(* Logix 5000 project; controller STAT 1756-L72 rev 20.12; software revision 20.04; part 12 of 34 *)
(* tags used below, declared in another part *)
   B10 : DINT[20];
   B14 : DINT[30];
   B16 : DINT[30];
   B17 : DINT[30];
   B3 : DINT[256];
   B9 : DINT[40];
   DateTime : DINT[7];   // DINT array tag for retrieve wallclock time through GSV created during conversion
   F8 : REAL[256];
   I10_000_Bit07 : ALIAS FOR I10[0].7;   // Hand Automaat CL8
   I10_000_Bit08 : ALIAS FOR I10[0].8;   // Drukknop start CL8 P 20
   I10_000_Bit09 : ALIAS FOR I10[0].9;   // Drukknop stop CL8 P 20
   I19_000_Bit02 : ALIAS FOR I19[0].2;   // vanne pmp puit 3 ouverte
   I19_000_Bit03 : ALIAS FOR I19[0].3;   // vanne pmp puit 3 fermee
   I19_000_Bit04 : ALIAS FOR I19[0].4;   // vanne pmp puit 2 ouverte
   I19_000_Bit05 : ALIAS FOR I19[0].5;   // vanne pmp puit 2 fermee
   I1_005_Bit15 : ALIAS FOR I1[5].15;
   I1_008_Bit01 : ALIAS FOR I1[8].1;   // Hand Automaat stormbekken
   I2_000_Bit04 : ALIAS FOR I2[0].4;   // Deelnoodstop cl6 eurowater
   I2_000_Bit05 : ALIAS FOR I2[0].5;   // Deelnoodstop cl7 IBT A
   I2_000_Bit07 : ALIAS FOR I2[0].7;   // Deelnoodstop cl7 IBT C
   I4_000_Bit00 : ALIAS FOR I4[0].0;   // Motor P3 voedingspomp in lijn
   I4_000_Bit03 : ALIAS FOR I4[0].3;   // Thermische storing voedingspomp fabriek 2
   I4_000_Bit04 : ALIAS FOR I4[0].4;   // Motor p4 in lijn in
   I4_000_Bit05 : ALIAS FOR I4[0].5;   // ready drive p4
   I4_000_Bit06 : ALIAS FOR I4[0].6;   // defaut drive P4
   I4_000_Bit11 : ALIAS FOR I4[0].11;   // pomp p23 in kelderkuip in dienst
   I5_001_Bit15 : ALIAS FOR I5[1].15;   // EV7_OPEN
   I6_000_Bit03 : ALIAS FOR I6[0].3;   // TH pmp PUT 2
   I6_000_Bit04 : ALIAS FOR I6[0].4;   // TH PMP PUT over
   I6_000_Bit05 : ALIAS FOR I6[0].5;   // th PMP PUT 1
   I6_000_Bit06 : ALIAS FOR I6[0].6;   // non existant th pmp 1 vijver
   I6_001_Bit04 : ALIAS FOR I6[1].4;   // niveau silo disolvent
   I7_000_Bit07 : ALIAS FOR I7[0].7;   // hoog alarm ketel tampon
   I7_000_Bit10 : ALIAS FOR I7[0].10;   // zeer hoog alarm ketel clarifee
   I7_000_Bit11 : ALIAS FOR I7[0].11;   // hoog zeer hoog alarm ketel clarifee
   I7_000_Bit12 : ALIAS FOR I7[0].12;   // laag alarm ketel clarifee
   I7_000_Bit13 : ALIAS FOR I7[0].13;   // zeer laag alarm ketel clarifee
   I7_001_Bit00 : ALIAS FOR I7[1].0;   // lus 4 niveau ketel clarifiee kontakt 3
   I9_000_Bit09 : ALIAS FOR I9[0].9;   // Hand_Auto CL7
   I9_000_Bit12 : ALIAS FOR I9[0].12;   // Drukknop start CL7 P4
   I9_000_Bit13 : ALIAS FOR I9[0].13;   // Drukknop stop CL7 P4
   I9_001_Bit00 : ALIAS FOR I9[1].0;   // Drukknop start CL7 P6
   I9_001_Bit01 : ALIAS FOR I9[1].1;   // Drukknop stop CL7 P6
   MW : BOOL;
   N11 : DINT[150];
   N12 : DINT[230];
   N13 : DINT[230];
   N7 : DINT[255];
   O12_000_Bit00 : ALIAS FOR O12[0].0;   // spoelpomp filters dubbele media P6_SPOEL
   O12_000_Bit12 : ALIAS FOR O12[0].12;   // Motor P19a zuiveringspomp controleweger P19_ZUIVERP
   O12_000_Bit13 : ALIAS FOR O12[0].13;   // Motor P20 zuiveringspomp controleweger P20_ZUIVERP
   O12_001_Bit03 : ALIAS FOR O12[1].3;   // Motor P7 voedingspomp omgekeerde osmose 1 P7_OSMOSE_1
   O12_001_Bit04 : ALIAS FOR O12[1].4;   // Motor P8 voedingspomp omgekeerde osmose 2 P8_OSMOSE_2
   O12_001_Bit05 : ALIAS FOR O12[1].5;   // Motor P9 voedingspomp omgekeerde osmose 3 P9_OSMOSE_3
   O15_001_Bit06 : ALIAS FOR O15[1].6;   // EV2 EV2
   O15_001_Bit11 : ALIAS FOR O15[1].11;   // EV7 EV7
   O16_000_Bit01 : ALIAS FOR O16[0].1;   // vanne pmp puit 3
   O16_000_Bit02 : ALIAS FOR O16[0].2;   // vanne pmp puit 2
   O18_001_Bit00 : ALIAS FOR O18[1].0;   // pompe 1 puisard ligne 4
   O18_001_Bit01 : ALIAS FOR O18[1].1;   // pompe 2 puisard ligne 4
   O18_001_Bit02 : ALIAS FOR O18[1].2;   // pmp put 2
   O18_001_Bit03 : ALIAS FOR O18[1].3;   // PMP PUT over
   O18_001_Bit04 : ALIAS FOR O18[1].4;   // PMP PUT 1
   O18_001_Bit05 : ALIAS FOR O18[1].5;   // pmp vijver IWM
   O18_001_Bit07 : ALIAS FOR O18[1].7;   // pomp pompen uit kelder p23
   O18_001_Bit08 : ALIAS FOR O18[1].8;   // pomp pompen uit kelder p24
   O1_006_Bit15 : ALIAS FOR O1[6].15;
   O27_000 : ALIAS FOR O27[0];
   O27_001 : ALIAS FOR O27[1];
   P4 : BOOL;
   Q2 : REAL;
   SCP_SPEED_PMP_FAB : SCP;
   SPEED_P3 : DINT;
   t1 : TIMER;
   T27 : TIMER[100];
   T4 : TIMER[200];
(* ibt, continued *)

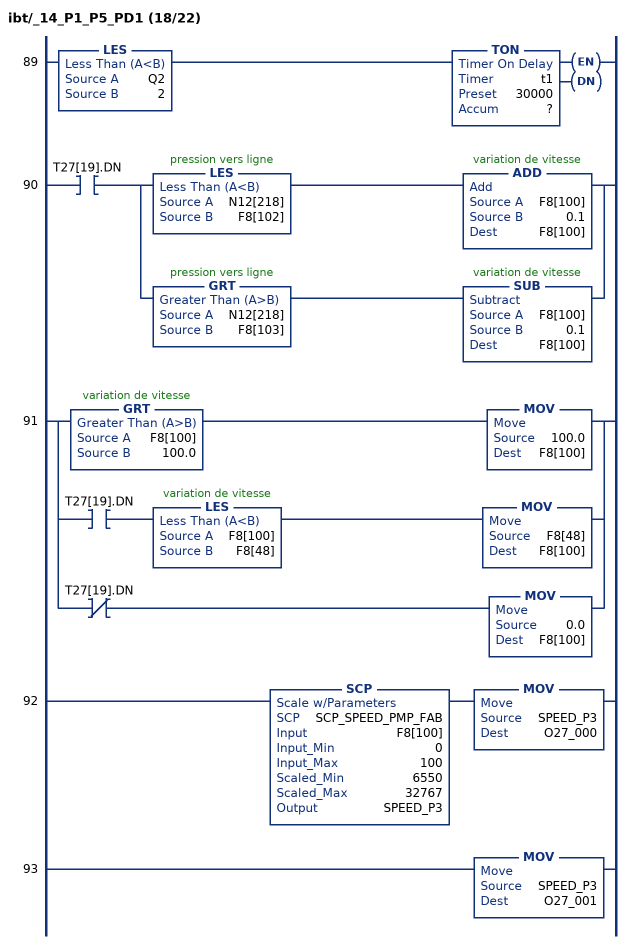
   [picture p178: ibt/_14_P1_P5_PD1 rungs 89-93]
   89: LES(Q2,2)TON(t1,?,?);
   90: XIC(T27[19].DN)[LES(N12[218],F8[102]) ADD(F8[100],0.1,F8[100]) ,GRT(N12[218],F8[103]) SUB(F8[100],0.1,F8[100]) ];
   91: [GRT(F8[100],100.0) MOV(100.0,F8[100]) ,XIC(T27[19].DN) LES(F8[100],F8[48]) MOV(F8[48],F8[100]) ,XIO(T27[19].DN) MOV(0.0,F8[100]) ];
   92: SCP(SCP_SPEED_PMP_FAB,F8[100],0,100,6550,32767,SPEED_P3)MOV(SPEED_P3,O27_000);
   93: MOV(SPEED_P3,O27_001);
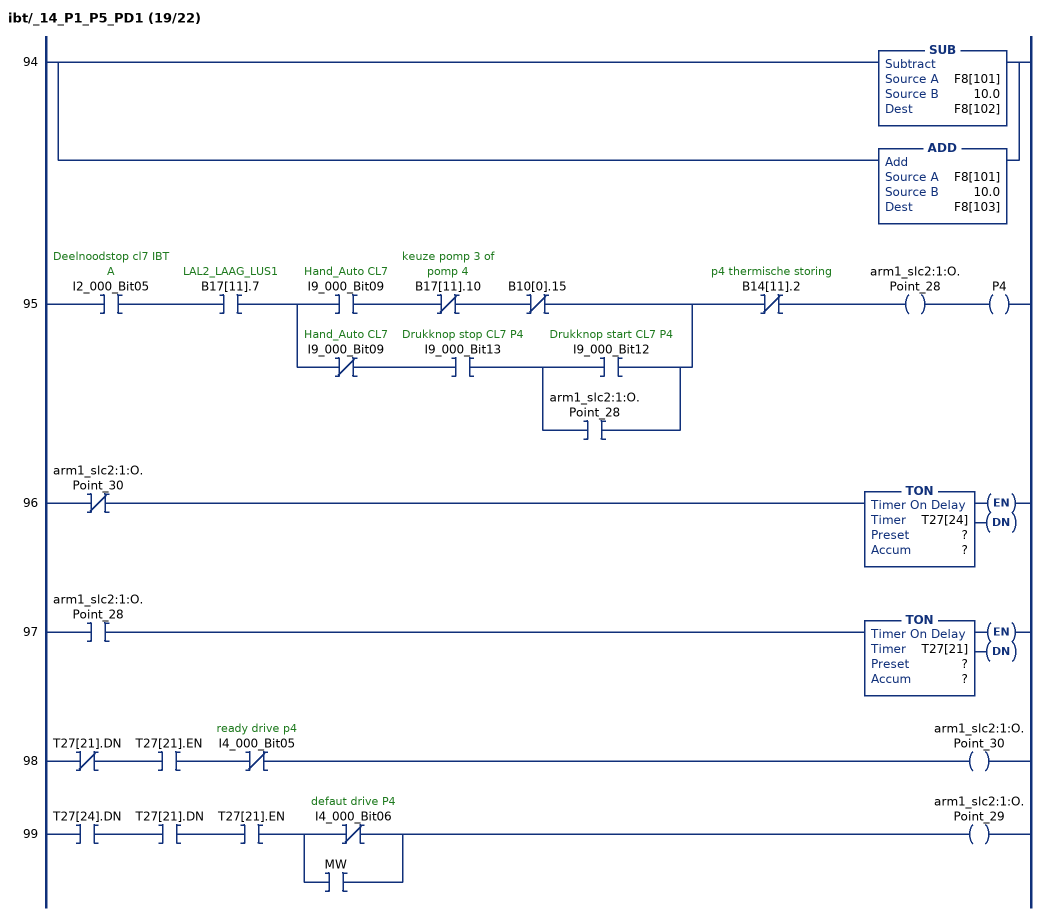
   94: [SUB(F8[101],10.0,F8[102]) ,ADD(F8[101],10.0,F8[103]) ];
   95: XIC(I2_000_Bit05)XIC(B17[11].7)[XIC(I9_000_Bit09) XIO(B17[11].10) XIO(B10[0].15) ,XIO(I9_000_Bit09) XIC(I9_000_Bit13) [XIC(I9_000_Bit12) ,XIC(arm1_slc2:1:O.Point_28) ] ]XIO(B14[11].2)OTE(arm1_slc2:1:O.Point_28)OTE(P4);
   96: XIO(arm1_slc2:1:O.Point_30)TON(T27[24],?,?);
   97: XIC(arm1_slc2:1:O.Point_28)TON(T27[21],?,?);
   98: XIO(T27[21].DN)XIC(T27[21].EN)XIO(I4_000_Bit05)OTE(arm1_slc2:1:O.Point_30);
   99: XIC(T27[24].DN)XIC(T27[21].DN)XIC(T27[21].EN)[XIO(I4_000_Bit06) ,XIC(MW) ]OTE(arm1_slc2:1:O.Point_29);
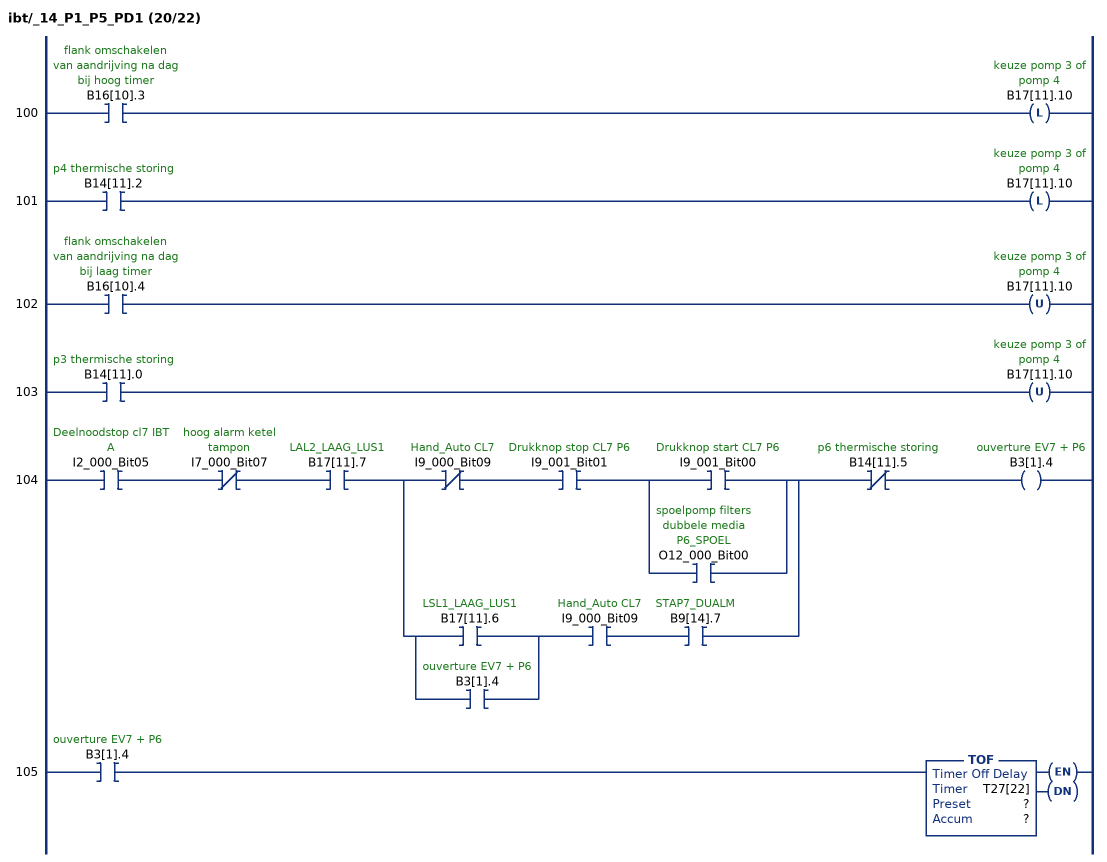
   100: XIC(B16[10].3)OTL(B17[11].10);
   101: XIC(B14[11].2)OTL(B17[11].10);
   102: XIC(B16[10].4)OTU(B17[11].10);
   103: XIC(B14[11].0)OTU(B17[11].10);
   104: XIC(I2_000_Bit05)XIO(I7_000_Bit07)XIC(B17[11].7)[XIO(I9_000_Bit09) XIC(I9_001_Bit01) [XIC(I9_001_Bit00) ,XIC(O12_000_Bit00) ] ,[XIC(B17[11].6) ,XIC(B3[1].4) ] XIC(I9_000_Bit09) XIC(B9[14].7) ]XIO(B14[11].5)OTE(B3[1].4);
   105: XIC(B3[1].4)TOF(T27[22],?,?);
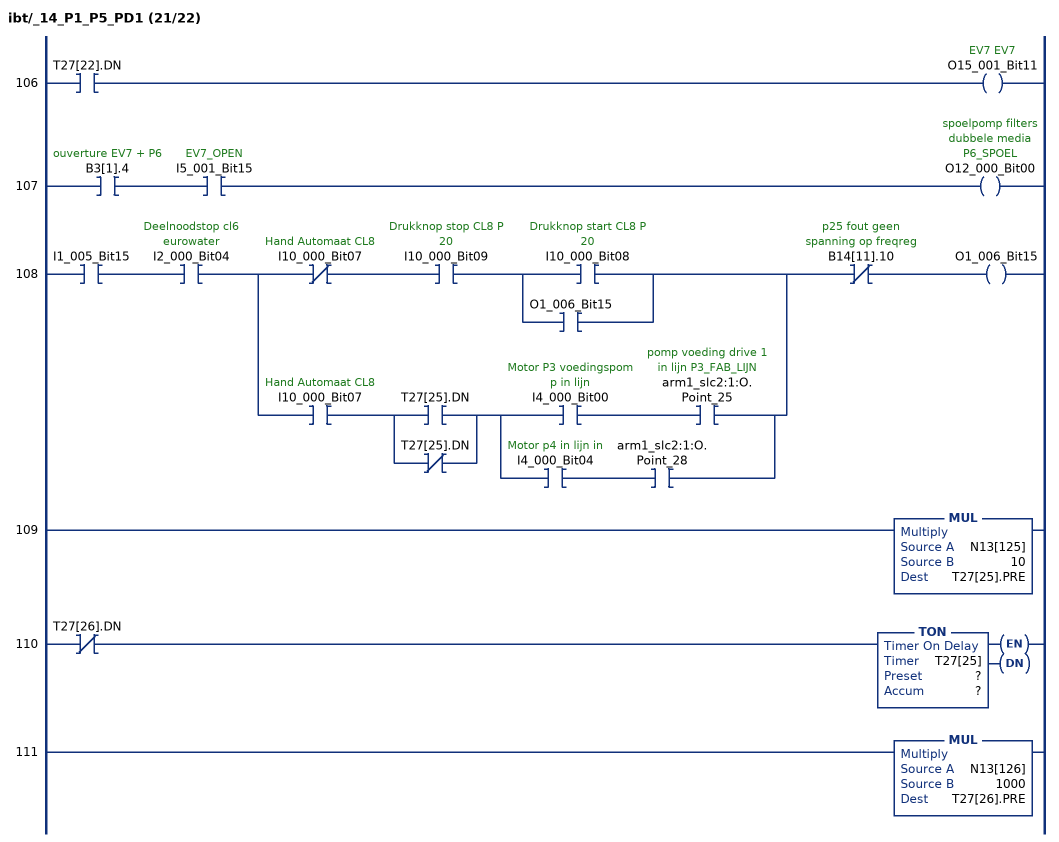
   106: XIC(T27[22].DN)OTE(O15_001_Bit11);
   107: XIC(B3[1].4)XIC(I5_001_Bit15)OTE(O12_000_Bit00);
   108: XIC(I1_005_Bit15)XIC(I2_000_Bit04)[XIO(I10_000_Bit07) XIC(I10_000_Bit09) [XIC(I10_000_Bit08) ,XIC(O1_006_Bit15) ] ,XIC(I10_000_Bit07) [XIC(T27[25].DN) ,XIO(T27[25].DN) ] [XIC(I4_000_Bit00) XIC(arm1_slc2:1:O.Point_25) ,XIC(I4_000_Bit04) XIC(arm1_slc2:1:O.Point_28) ] ]XIO(B14[11].10)OTE(O1_006_Bit15);
   109: MUL(N13[125],10,T27[25].PRE);
   110: XIO(T27[26].DN)TON(T27[25],?,?);
   111: MUL(N13[126],1000,T27[26].PRE);
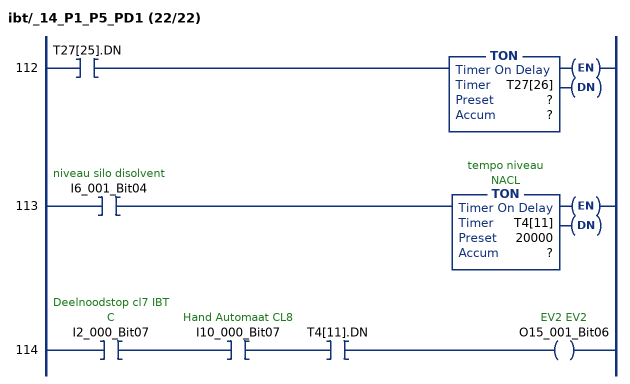
   112: XIC(T27[25].DN)TON(T27[26],?,?);
   113: XIC(I6_001_Bit04)TON(T4[11],?,?);
   114: XIC(I2_000_Bit07)XIC(I10_000_Bit07)XIC(T4[11].DN)OTE(O15_001_Bit06);
END_ROUTINE

ROUTINE _15_PMP_PUISAR   (* ladder *)
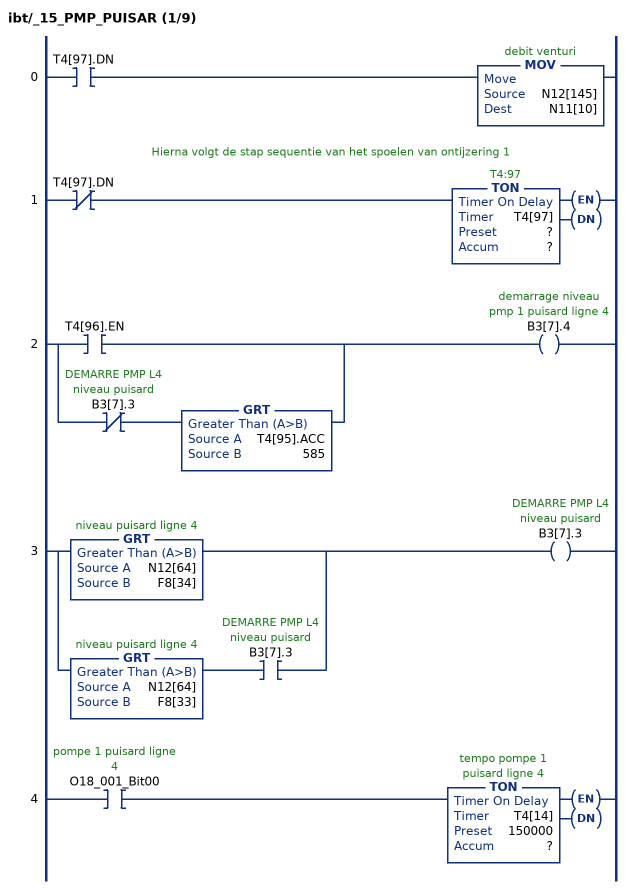
   0: XIC(T4[97].DN)MOV(N12[145],N11[10]);
   // Hierna volgt de stap sequentie van het spoelen van ontijzering 1
   1: XIO(T4[97].DN)TON(T4[97],?,?);
   2: [XIC(T4[96].EN) ,XIO(B3[7].3) GRT(T4[95].ACC,585) ]OTE(B3[7].4);
   3: [GRT(N12[64],F8[34]) ,GRT(N12[64],F8[33]) XIC(B3[7].3) ]OTE(B3[7].3);
   4: XIC(O18_001_Bit00)TON(T4[14],?,?);
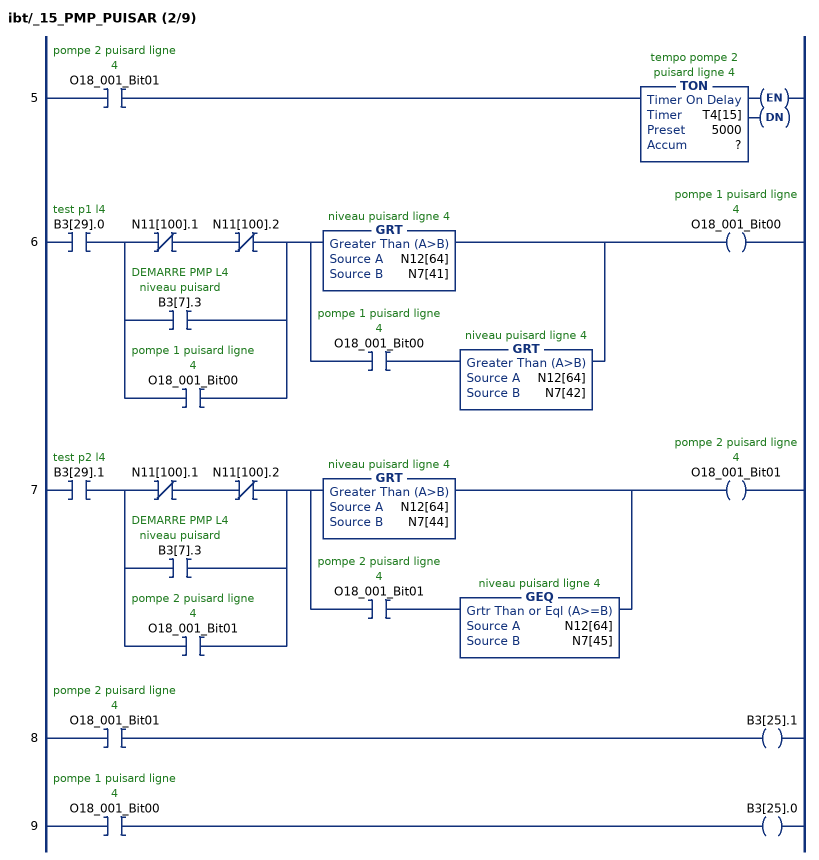
   5: XIC(O18_001_Bit01)TON(T4[15],?,?);
   6: XIC(B3[29].0)[XIO(N11[100].1) XIO(N11[100].2) ,XIC(B3[7].3) ,XIC(O18_001_Bit00) ][GRT(N12[64],N7[41]) ,XIC(O18_001_Bit00) GRT(N12[64],N7[42]) ]OTE(O18_001_Bit00);
   7: XIC(B3[29].1)[XIO(N11[100].1) XIO(N11[100].2) ,XIC(B3[7].3) ,XIC(O18_001_Bit01) ][GRT(N12[64],N7[44]) ,XIC(O18_001_Bit01) GEQ(N12[64],N7[45]) ]OTE(O18_001_Bit01);
   8: XIC(O18_001_Bit01)OTE(B3[25].1);
   9: XIC(O18_001_Bit00)OTE(B3[25].0);
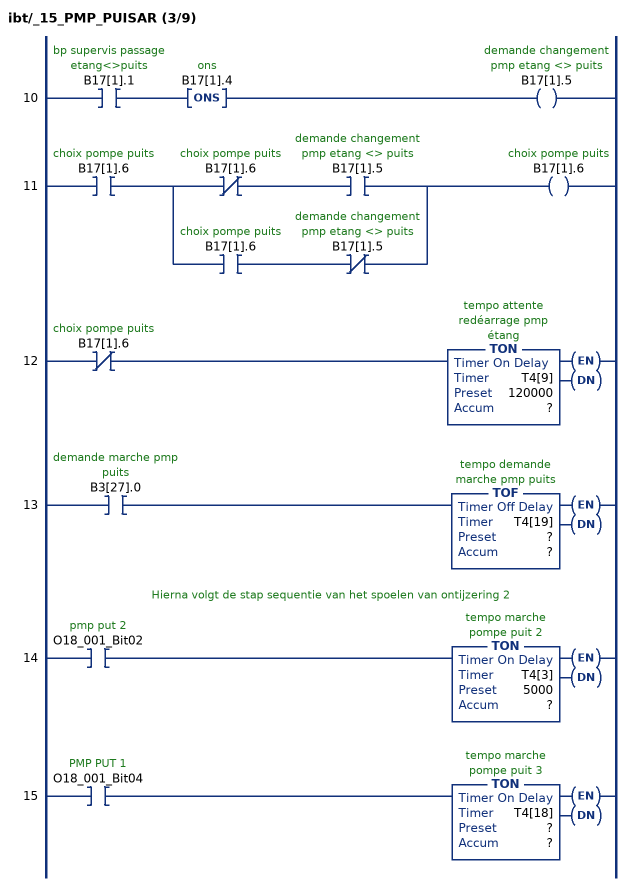
   10: XIC(B17[1].1)ONS(B17[1].4)OTE(B17[1].5);
   11: XIC(B17[1].6)[XIO(B17[1].6) XIC(B17[1].5) ,XIC(B17[1].6) XIO(B17[1].5) ]OTE(B17[1].6);
   12: XIO(B17[1].6)TON(T4[9],?,?);
   13: XIC(B3[27].0)TOF(T4[19],?,?);
   // Hierna volgt de stap sequentie van het spoelen van ontijzering 2
   14: XIC(O18_001_Bit02)TON(T4[3],?,?);
   15: XIC(O18_001_Bit04)TON(T4[18],?,?);
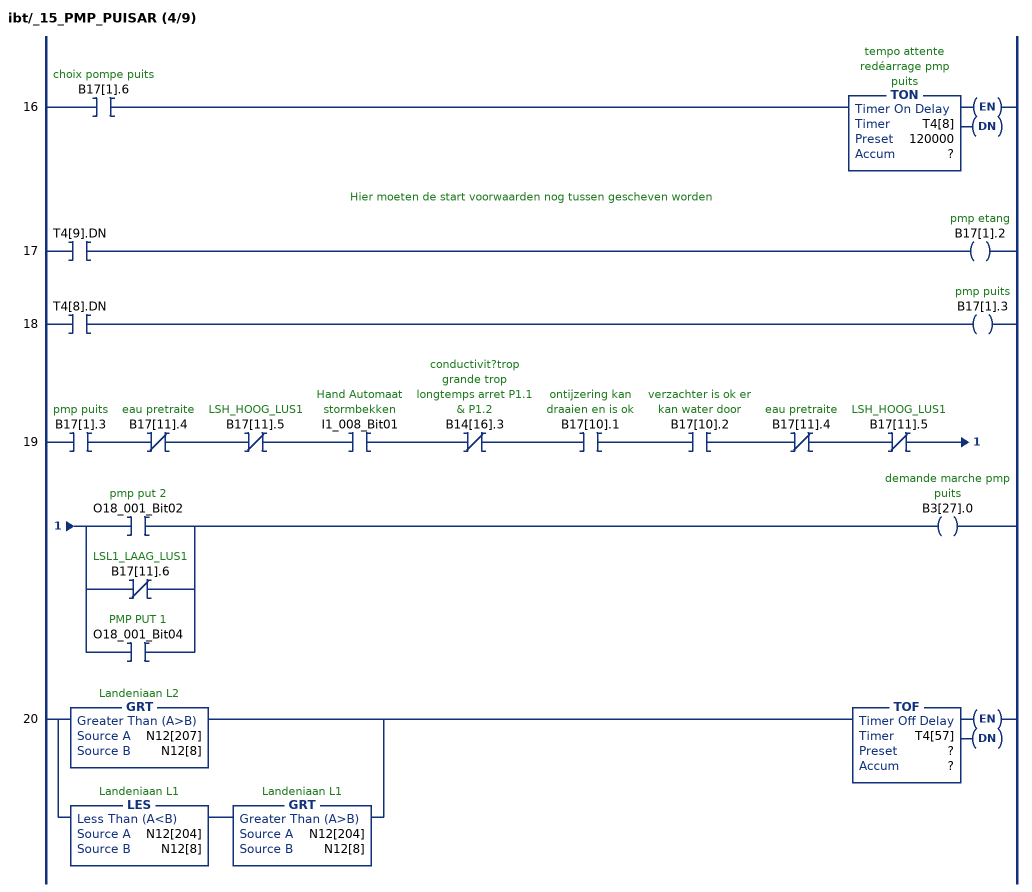
   16: XIC(B17[1].6)TON(T4[8],?,?);
   // Hier moeten de start voorwaarden nog tussen gescheven worden
   17: XIC(T4[9].DN)OTE(B17[1].2);
   18: XIC(T4[8].DN)OTE(B17[1].3);
   19: XIC(B17[1].3)XIO(B17[11].4)XIO(B17[11].5)XIC(I1_008_Bit01)XIO(B14[16].3)XIC(B17[10].1)XIC(B17[10].2)XIO(B17[11].4)XIO(B17[11].5)[XIC(O18_001_Bit02) ,XIO(B17[11].6) ,XIC(O18_001_Bit04) ]OTE(B3[27].0);
   20: [GRT(N12[207],N12[8]) ,LES(N12[204],N12[8]) GRT(N12[204],N12[8]) ]TOF(T4[57],?,?);
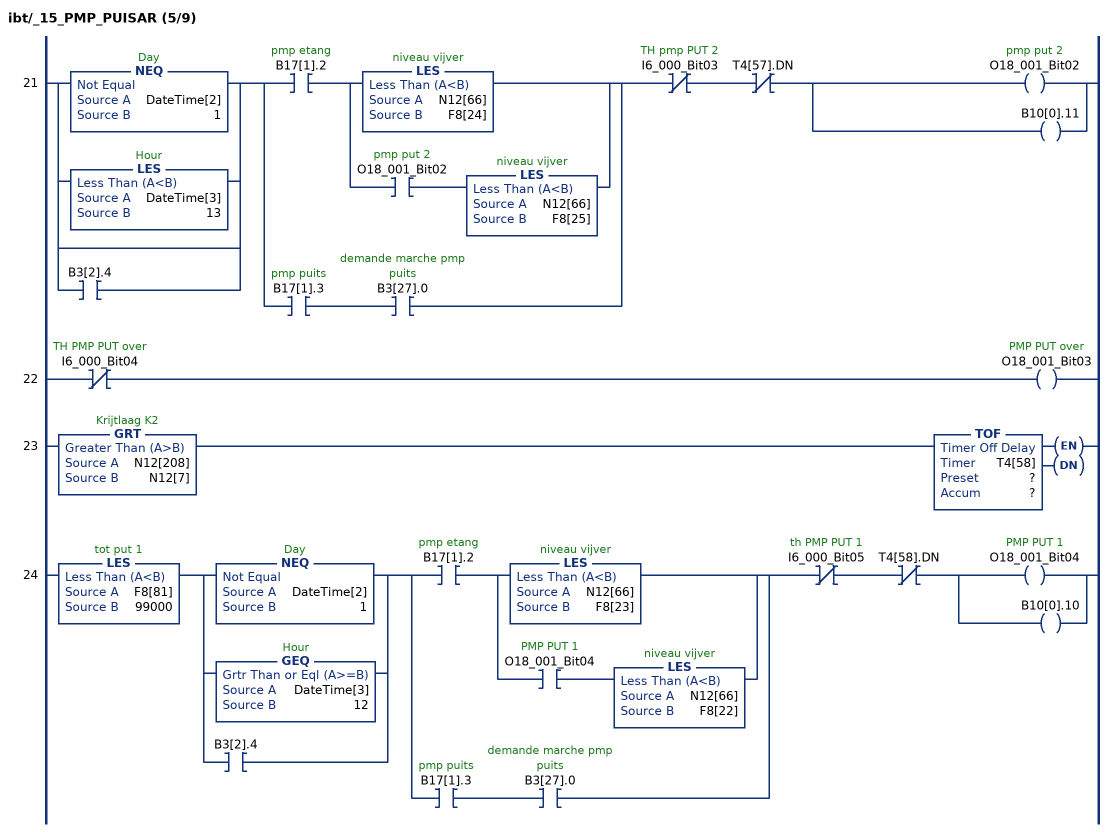
   21: [NEQ(DateTime[2],1) ,LES(DateTime[3],13) ,,XIC(B3[2].4) ][XIC(B17[1].2) [LES(N12[66],F8[24]) ,XIC(O18_001_Bit02) LES(N12[66],F8[25]) ] ,XIC(B17[1].3) XIC(B3[27].0) ]XIO(I6_000_Bit03)XIO(T4[57].DN)[OTE(O18_001_Bit02) ,OTE(B10[0].11) ];
   22: XIO(I6_000_Bit04)OTE(O18_001_Bit03);
   23: GRT(N12[208],N12[7])TOF(T4[58],?,?);
   24: LES(F8[81],99000)[NEQ(DateTime[2],1) ,GEQ(DateTime[3],12) ,XIC(B3[2].4) ][XIC(B17[1].2) [LES(N12[66],F8[23]) ,XIC(O18_001_Bit04) LES(N12[66],F8[22]) ] ,XIC(B17[1].3) XIC(B3[27].0) ]XIO(I6_000_Bit05)XIO(T4[58].DN)[OTE(O18_001_Bit04) ,OTE(B10[0].10) ];
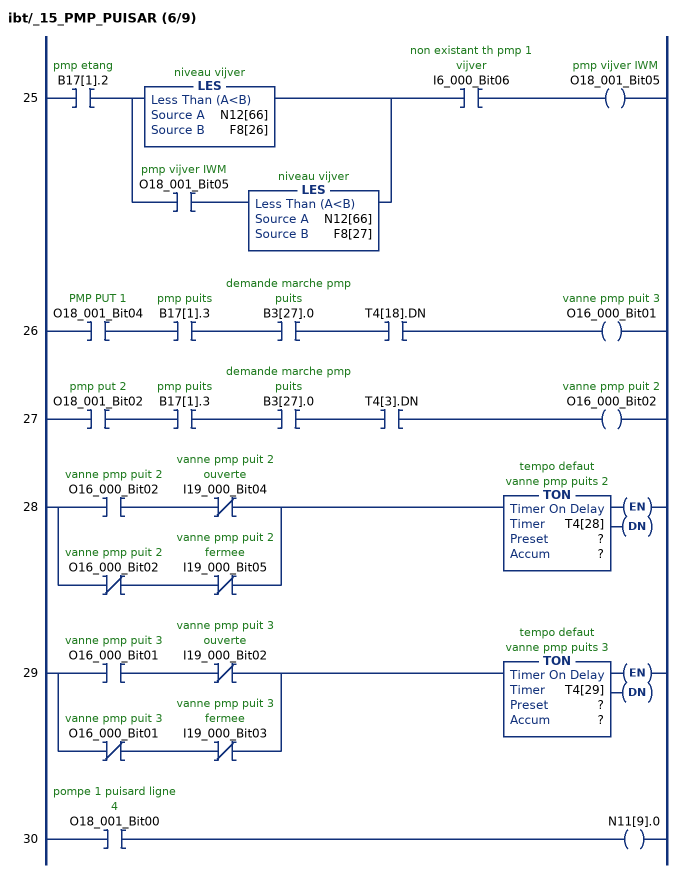
   25: XIC(B17[1].2)[LES(N12[66],F8[26]) ,XIC(O18_001_Bit05) LES(N12[66],F8[27]) ]XIC(I6_000_Bit06)OTE(O18_001_Bit05);
   26: XIC(O18_001_Bit04)XIC(B17[1].3)XIC(B3[27].0)XIC(T4[18].DN)OTE(O16_000_Bit01);
   27: XIC(O18_001_Bit02)XIC(B17[1].3)XIC(B3[27].0)XIC(T4[3].DN)OTE(O16_000_Bit02);
   28: [XIC(O16_000_Bit02) XIO(I19_000_Bit04) ,XIO(O16_000_Bit02) XIO(I19_000_Bit05) ]TON(T4[28],?,?);
   29: [XIC(O16_000_Bit01) XIO(I19_000_Bit02) ,XIO(O16_000_Bit01) XIO(I19_000_Bit03) ]TON(T4[29],?,?);
   30: XIC(O18_001_Bit00)OTE(N11[9].0);
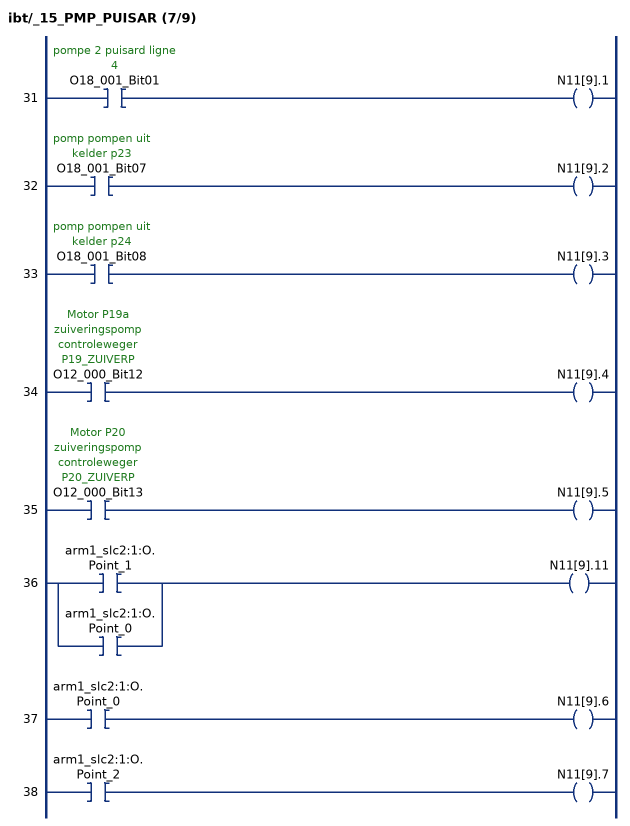
   31: XIC(O18_001_Bit01)OTE(N11[9].1);
   32: XIC(O18_001_Bit07)OTE(N11[9].2);
   33: XIC(O18_001_Bit08)OTE(N11[9].3);
   34: XIC(O12_000_Bit12)OTE(N11[9].4);
   35: XIC(O12_000_Bit13)OTE(N11[9].5);
   36: [XIC(arm1_slc2:1:O.Point_1) ,XIC(arm1_slc2:1:O.Point_0) ]OTE(N11[9].11);
   37: XIC(arm1_slc2:1:O.Point_0)OTE(N11[9].6);
   38: XIC(arm1_slc2:1:O.Point_2)OTE(N11[9].7);
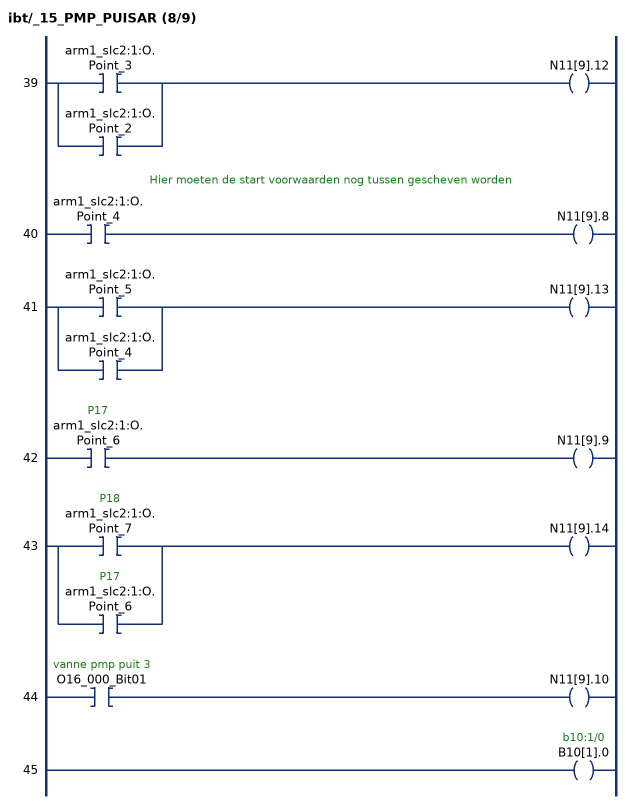
   39: [XIC(arm1_slc2:1:O.Point_3) ,XIC(arm1_slc2:1:O.Point_2) ]OTE(N11[9].12);
   // Hier moeten de start voorwaarden nog tussen gescheven worden
   40: XIC(arm1_slc2:1:O.Point_4)OTE(N11[9].8);
   41: [XIC(arm1_slc2:1:O.Point_5) ,XIC(arm1_slc2:1:O.Point_4) ]OTE(N11[9].13);
   42: XIC(arm1_slc2:1:O.Point_6)OTE(N11[9].9);
   43: [XIC(arm1_slc2:1:O.Point_7) ,XIC(arm1_slc2:1:O.Point_6) ]OTE(N11[9].14);
   44: XIC(O16_000_Bit01)OTE(N11[9].10);
   45: OTE(B10[1].0);
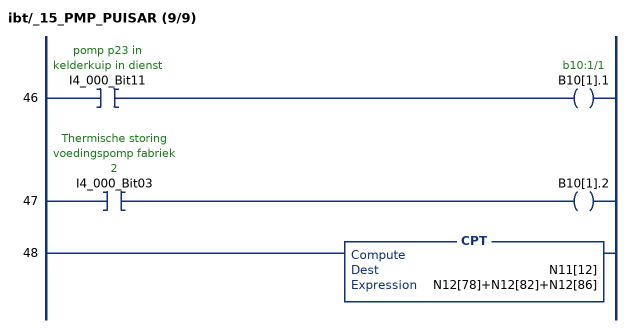
   46: XIC(I4_000_Bit11)OTE(B10[1].1);
   47: XIC(I4_000_Bit03)OTE(B10[1].2);
   48: CPT(N11[12],N12[78]+N12[82]+N12[86]);
END_ROUTINE

ROUTINE _16_ALI_OS_P19   (* ladder *)
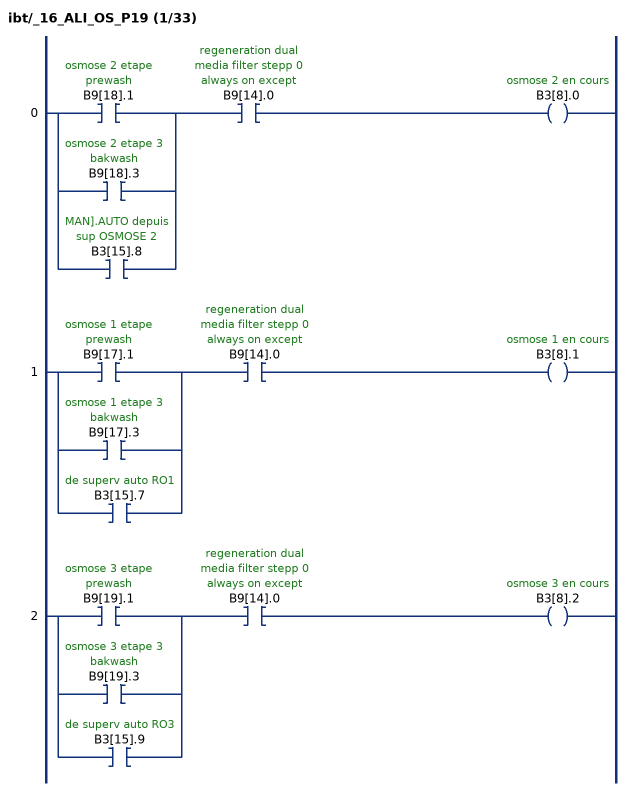
   0: [XIC(B9[18].1) ,XIC(B9[18].3) ,XIC(B3[15].8) ]XIC(B9[14].0)OTE(B3[8].0);
   1: [XIC(B9[17].1) ,XIC(B9[17].3) ,XIC(B3[15].7) ]XIC(B9[14].0)OTE(B3[8].1);
   2: [XIC(B9[19].1) ,XIC(B9[19].3) ,XIC(B3[15].9) ]XIC(B9[14].0)OTE(B3[8].2);
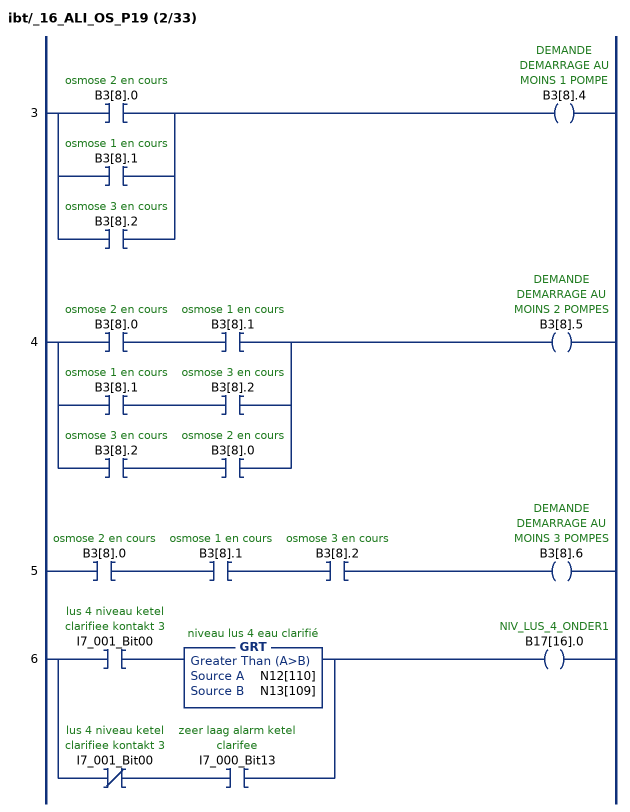
   3: [XIC(B3[8].0) ,XIC(B3[8].1) ,XIC(B3[8].2) ]OTE(B3[8].4);
   4: [XIC(B3[8].0) XIC(B3[8].1) ,XIC(B3[8].1) XIC(B3[8].2) ,XIC(B3[8].2) XIC(B3[8].0) ]OTE(B3[8].5);
   5: XIC(B3[8].0)XIC(B3[8].1)XIC(B3[8].2)OTE(B3[8].6);
   6: [XIC(I7_001_Bit00) GRT(N12[110],N13[109]) ,XIO(I7_001_Bit00) XIC(I7_000_Bit13) ]OTE(B17[16].0);
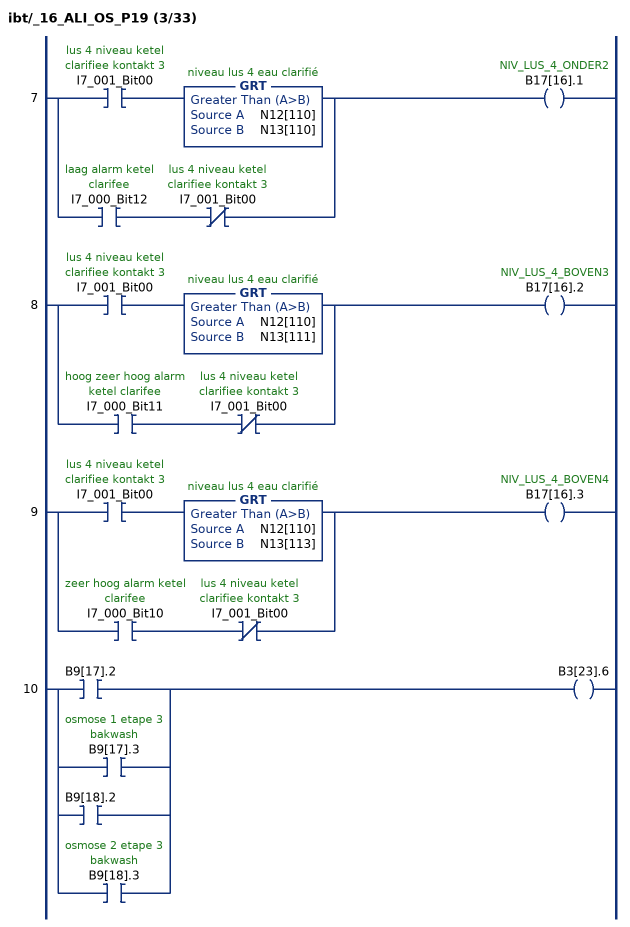
   7: [XIC(I7_001_Bit00) GRT(N12[110],N13[110]) ,XIC(I7_000_Bit12) XIO(I7_001_Bit00) ]OTE(B17[16].1);
   8: [XIC(I7_001_Bit00) GRT(N12[110],N13[111]) ,XIC(I7_000_Bit11) XIO(I7_001_Bit00) ]OTE(B17[16].2);
   9: [XIC(I7_001_Bit00) GRT(N12[110],N13[113]) ,XIC(I7_000_Bit10) XIO(I7_001_Bit00) ]OTE(B17[16].3);
   10: [XIC(B9[17].2) ,XIC(B9[17].3) ,XIC(B9[18].2) ,XIC(B9[18].3) ]OTE(B3[23].6);
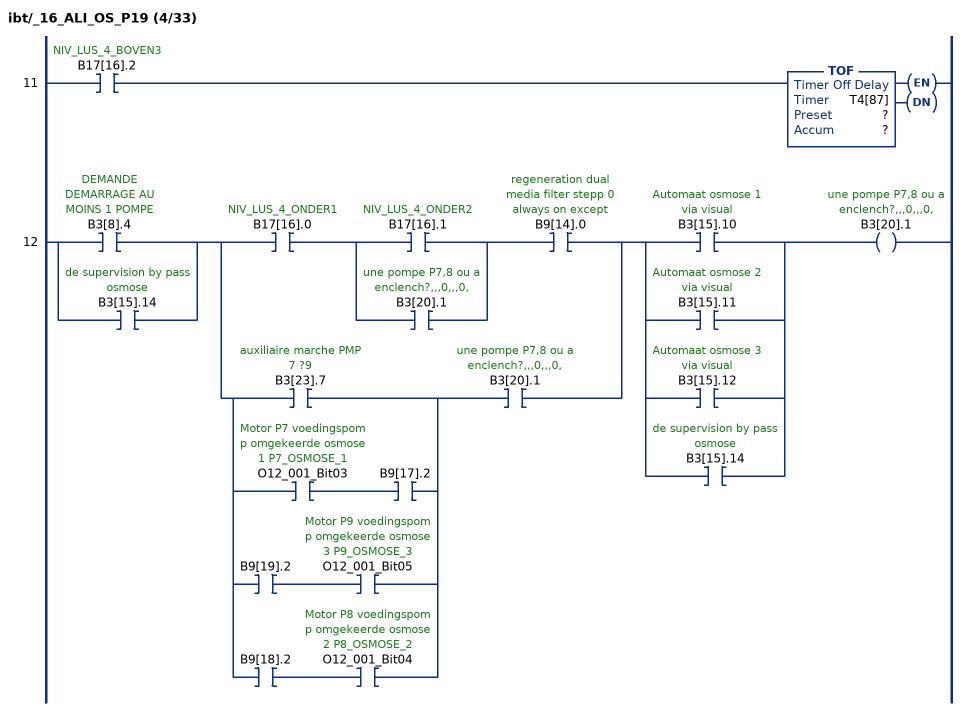
   11: XIC(B17[16].2)TOF(T4[87],?,?);
   12: [XIC(B3[8].4) ,XIC(B3[15].14) ][XIC(B17[16].0) [XIC(B17[16].1) ,XIC(B3[20].1) ] XIC(B9[14].0) ,[XIC(B3[23].7) ,XIC(O12_001_Bit03) XIC(B9[17].2) ,XIC(B9[19].2) XIC(O12_001_Bit05) ,XIC(B9[18].2) XIC(O12_001_Bit04) ] XIC(B3[20].1) ][XIC(B3[15].10) ,[XIC(B3[15].11) ,[XIC(B3[15].12) ,XIC(B3[15].14) ] ] ]OTE(B3[20].1);
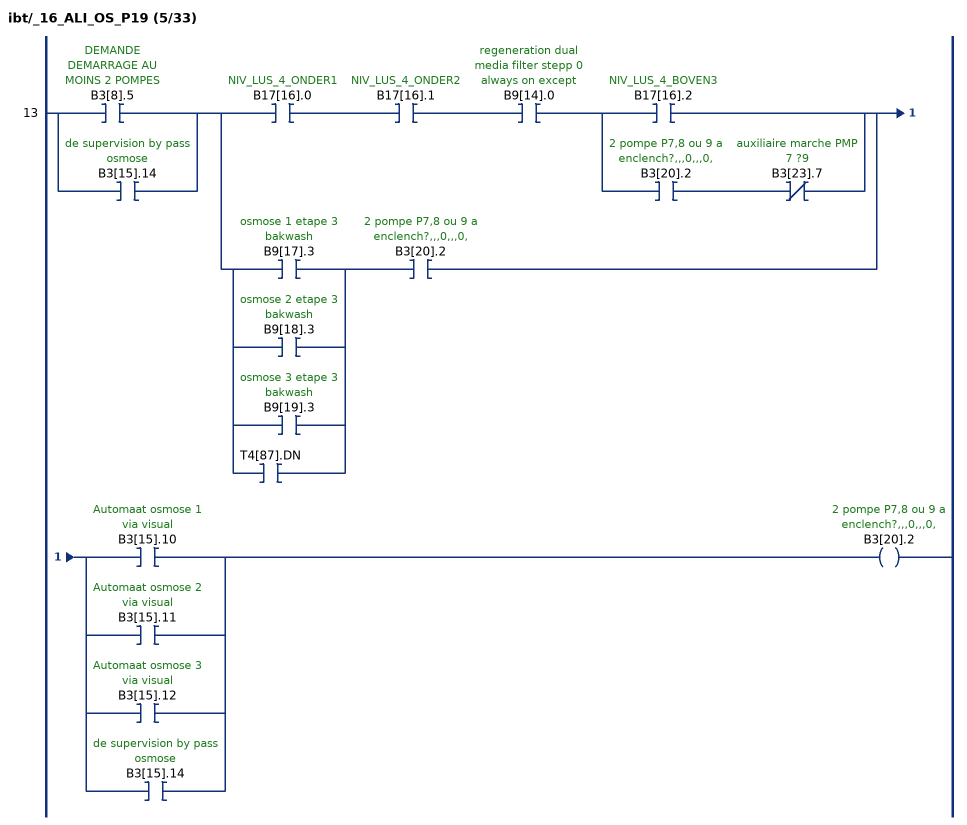
   13: [XIC(B3[8].5) ,XIC(B3[15].14) ][XIC(B17[16].0) XIC(B17[16].1) XIC(B9[14].0) [XIC(B17[16].2) ,XIC(B3[20].2) XIO(B3[23].7) ] ,[XIC(B9[17].3) ,XIC(B9[18].3) ,XIC(B9[19].3) ,XIC(T4[87].DN) ] XIC(B3[20].2) ][XIC(B3[15].10) ,[XIC(B3[15].11) ,[XIC(B3[15].12) ,XIC(B3[15].14) ] ] ]OTE(B3[20].2);
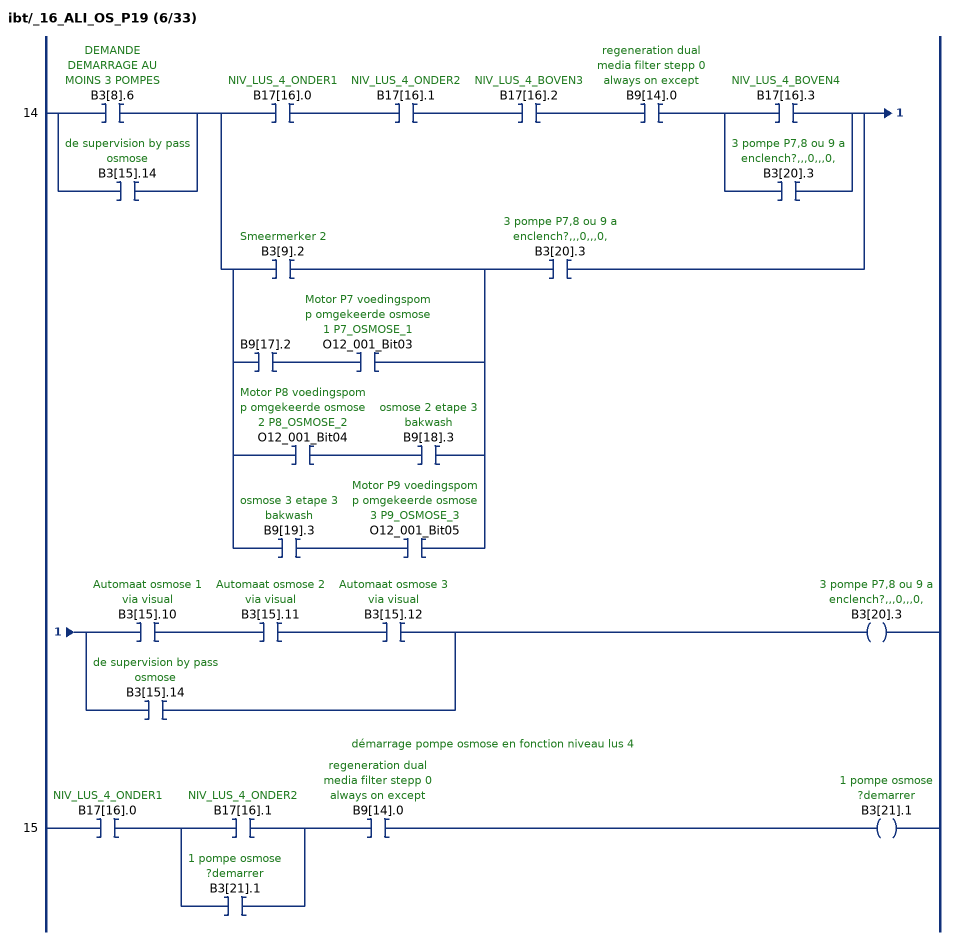
   14: [XIC(B3[8].6) ,XIC(B3[15].14) ][XIC(B17[16].0) XIC(B17[16].1) XIC(B17[16].2) XIC(B9[14].0) [XIC(B17[16].3) ,XIC(B3[20].3) ] ,[XIC(B3[9].2) ,[XIC(B9[17].2) XIC(O12_001_Bit03) ,[XIC(O12_001_Bit04) XIC(B9[18].3) ,XIC(B9[19].3) XIC(O12_001_Bit05) ] ] ] XIC(B3[20].3) ][XIC(B3[15].10) XIC(B3[15].11) XIC(B3[15].12) ,XIC(B3[15].14) ]OTE(B3[20].3);
   // démarrage pompe osmose en fonction niveau lus 4
   15: XIC(B17[16].0)[XIC(B17[16].1) ,XIC(B3[21].1) ]XIC(B9[14].0)OTE(B3[21].1);
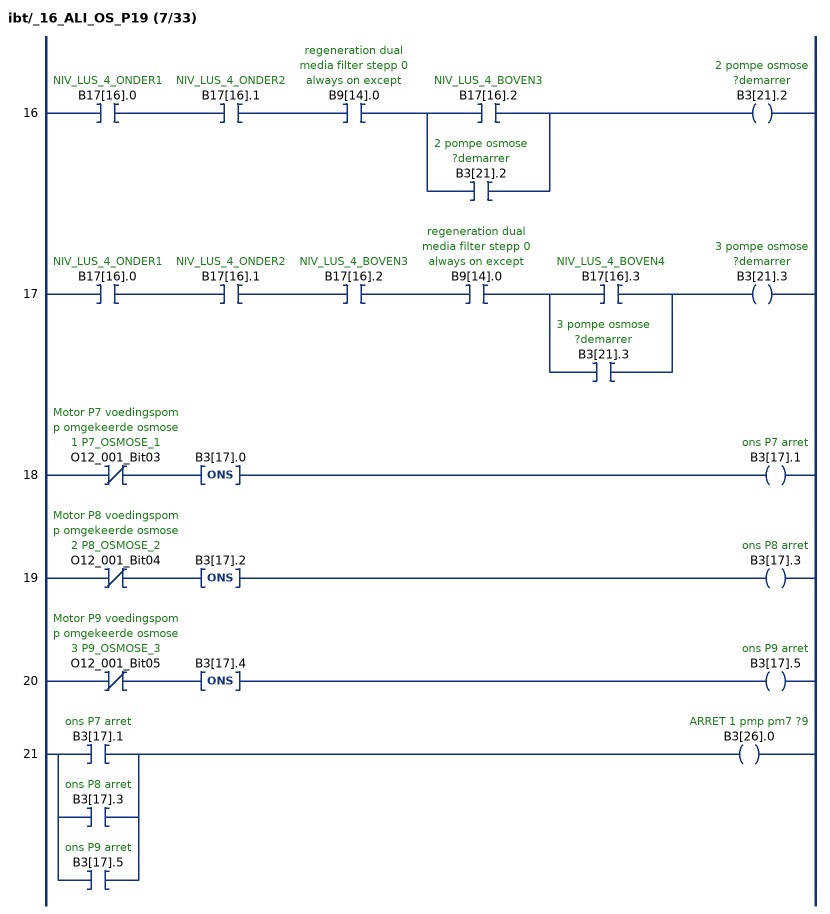
   16: XIC(B17[16].0)XIC(B17[16].1)XIC(B9[14].0)[XIC(B17[16].2) ,XIC(B3[21].2) ]OTE(B3[21].2);
   17: XIC(B17[16].0)XIC(B17[16].1)XIC(B17[16].2)XIC(B9[14].0)[XIC(B17[16].3) ,XIC(B3[21].3) ]OTE(B3[21].3);
   18: XIO(O12_001_Bit03)ONS(B3[17].0)OTE(B3[17].1);
   19: XIO(O12_001_Bit04)ONS(B3[17].2)OTE(B3[17].3);
   20: XIO(O12_001_Bit05)ONS(B3[17].4)OTE(B3[17].5);
   21: [XIC(B3[17].1) ,[XIC(B3[17].3) ,XIC(B3[17].5) ] ]OTE(B3[26].0);
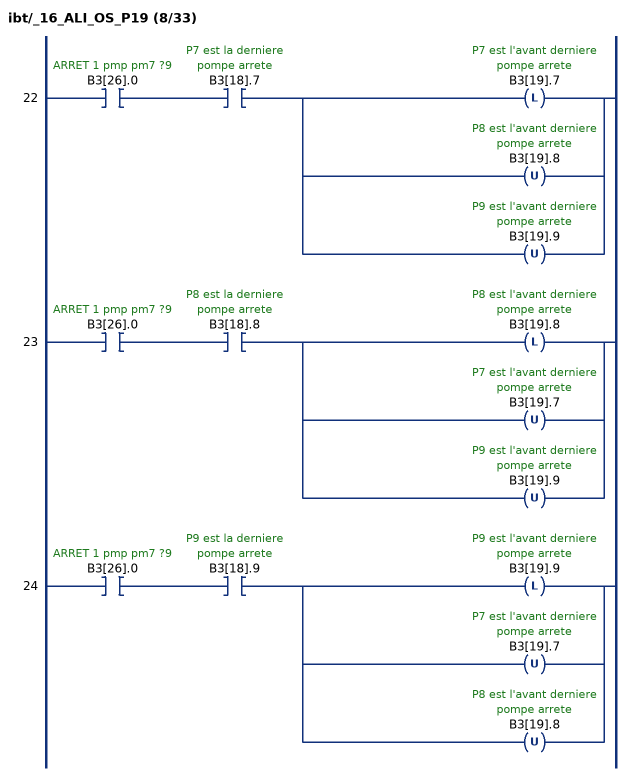
   22: XIC(B3[26].0)XIC(B3[18].7)[OTL(B3[19].7) ,[OTU(B3[19].8) ,OTU(B3[19].9) ] ];
   23: XIC(B3[26].0)XIC(B3[18].8)[OTL(B3[19].8) ,[OTU(B3[19].7) ,OTU(B3[19].9) ] ];
   24: XIC(B3[26].0)XIC(B3[18].9)[OTL(B3[19].9) ,[OTU(B3[19].7) ,OTU(B3[19].8) ] ];
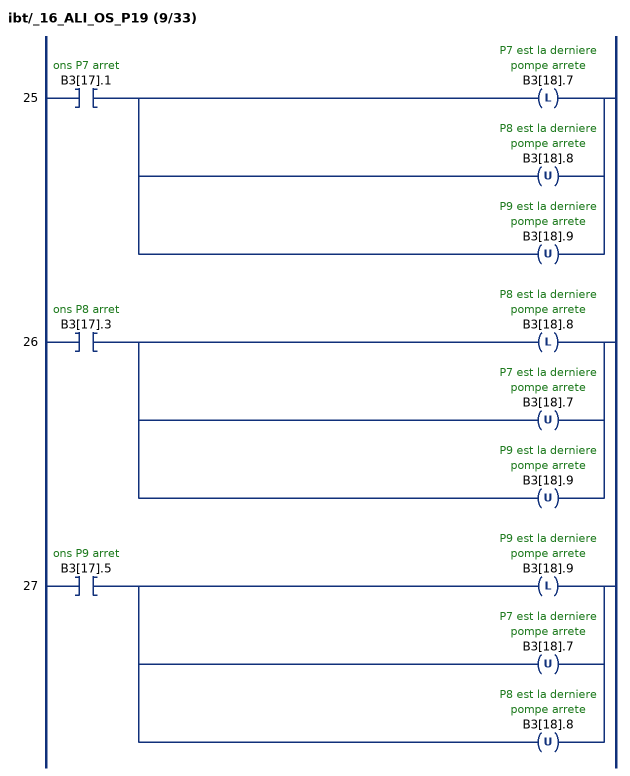
   25: XIC(B3[17].1)[OTL(B3[18].7) ,[OTU(B3[18].8) ,OTU(B3[18].9) ] ];
   26: XIC(B3[17].3)[OTL(B3[18].8) ,[OTU(B3[18].7) ,OTU(B3[18].9) ] ];
   27: XIC(B3[17].5)[OTL(B3[18].9) ,[OTU(B3[18].7) ,OTU(B3[18].8) ] ];
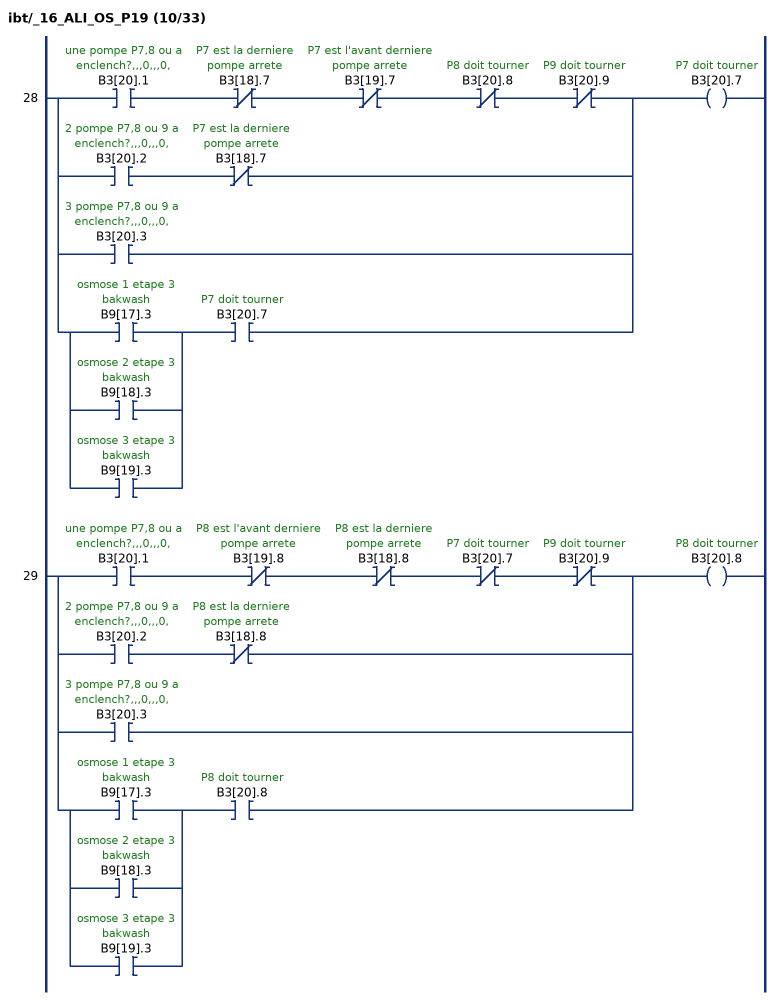
   28: [XIC(B3[20].1) XIO(B3[18].7) XIO(B3[19].7) XIO(B3[20].8) XIO(B3[20].9) ,[XIC(B3[20].2) XIO(B3[18].7) ,XIC(B3[20].3) ] ,[XIC(B9[17].3) ,XIC(B9[18].3) ,XIC(B9[19].3) ] XIC(B3[20].7) ]OTE(B3[20].7);
   29: [XIC(B3[20].1) XIO(B3[19].8) XIO(B3[18].8) XIO(B3[20].7) XIO(B3[20].9) ,[XIC(B3[20].2) XIO(B3[18].8) ,XIC(B3[20].3) ] ,[XIC(B9[17].3) ,XIC(B9[18].3) ,XIC(B9[19].3) ] XIC(B3[20].8) ]OTE(B3[20].8);
